FUNCTION_BLOCK Blinky (* Composite Function Block Type *)
  (* Standard: 61499-2; Description: Copyright (c) 2019 Jan Holzweber This program and the accompanying materials are made available under the terms of the Eclipse Public License 2.0 which is available at https://www.eclipse.org/legal/epl-2.0/ SPDX-License-Identifier: EPL-2.0 *)
  (* Version 1.0, 2019-07-18, Jan Holzweber *)
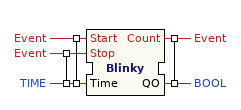
  EVENT_INPUT
    Start WITH Time;
    Stop WITH Time;
  END_EVENT
  EVENT_OUTPUT
    Count WITH QO;
  END_EVENT
  VAR_INPUT
    Time : TIME;
  END_VAR
  VAR_OUTPUT
    QO : BOOL;
  END_VAR
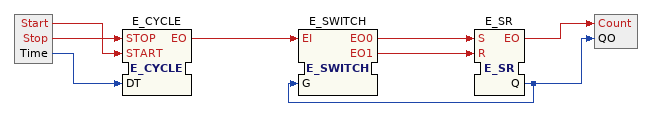
  FBS
    E_CYCLE : E_CYCLE;
    E_SWITCH : E_SWITCH;
    E_SR : E_SR;
  END_FBS
  EVENT_CONNECTIONS
    E_CYCLE.EO TO E_SWITCH.EI;
    E_SWITCH.EO0 TO E_SR.S;
    E_SWITCH.EO1 TO E_SR.R;
    E_SR.EO TO Count;
    Stop TO E_CYCLE.STOP;
    Start TO E_CYCLE.START;
  END_CONNECTIONS
  DATA_CONNECTIONS
    E_SR.Q TO QO;
    E_SR.Q TO E_SWITCH.G;
    Time TO E_CYCLE.DT;
  END_CONNECTIONS
END_FUNCTION_BLOCK
